// TIA Portal V18 export
// export: Created 2025-12-01T12:39:35.7160245Z, ExportSetting None, DisplayName Totally Integrated Automation Portal, DisplayVersion V18 Update 5, DisplayName TIA Portal Openness, DisplayVersion V18 Update 5, DisplayName TIA Portal Teamcenter Gateway, DisplayVersion V18, DisplayName TIA Portal Version Control Interface, DisplayVersion V18, DisplayName STEP 7 Professional, DisplayVersion V18 Update 5, DisplayName STEP 7 Safety, DisplayVersion V18, DisplayName WinCC Professional, DisplayVersion V18 Update 5
VAR_GLOBAL   // PLC tag table "RFID"
END_VAR
VAR_GLOBAL CONSTANT   // user constants
   OP220_RFID初始化 : Int := 99;   // OP220_RFID初始化
   OP220_RFID读取 : Int := 1;   // OP220_RFID读取
   OP220_RFID写入 : Int := 2;   // OP220_RFID写入
   OP220_RFID自动正常循环模式 : USInt := 0;   // OP220_RFID自动正常循环模式
   OP220_RFID返工模式 : USInt := 1;   // OP220_RFID返工模式
   OP220_RFID清线模式 : USInt := 2;   // OP220_RFID清线模式
   OP220_RFID自动空循环模式 : USInt := 3;   // OP220_RFID自动空循环模式
   OP220_RFID空托盘循环模式 : USInt := 4;   // OP220_RFID空托盘循环模式
   OP220_RFID换型托盘模式 : USInt := 5;   // OP220_RFID换型托盘模式
   OP220_RFID校验托盘模式 : USInt := 6;   // OP220_RFID校验托盘模式
END_VAR
